FUNCTION F_AlyTimestampToFileTime : ULINT
VAR_INPUT
	tTimestamp: ULINT;
END_VAR
VAR
	tFileTime: T_FILETIME;
	
	fbToUTC: FB_TzSpecificLocalTimeToFileTime;
	//Malay Peninsula Daylight Time
	//(UTC+08:00) Kuala Lumpur, Singapore
	tzInfo: ST_TimeZoneInformation := (bias := -480);
END_VAR

tFileTime:= DCTIME64_TO_Filetime(tTimestamp);

fbToUTC(in:= tFileTime, tzInfo:= tzInfo);
F_AlyTimestampToFileTime:= ULARGE_TO_ULINT(ULARGE_INTEGER(fbToUTC.out.dwHighDateTime, fbToUTC.out.dwLowDateTime));

END_FUNCTION

(* stored: POU F_AlyTimestampToFileTime: Id 0eab0d49-8c9d-4c06-ad36-5c00ac5da2b6, SpecialFunc None *)
